// TIA Portal V20 export
ORGANIZATION_BLOCK "Startup"   // OB1020, LAD, Startup
TITLE = "Complete Restart"
AUTHOR : ERsystem_FA2_DH. Kim
// stored: AutoNumber false, IsIECCheckEnabled true, Namespace Unit1.Em2, SetENOAutomatically false
   VAR_INPUT
      LostRetentive : Bool;   // True if retentive data are lost
      LostRTC : Bool;   // True if date and time are lost
   END_VAR
BEGIN

REGION Network 1 (SCL): Build the Absolut Reference Designator
   // Set the Absoult Reference Designator in the Config DB
   IF LEN(IN := "Unit1.Em2.Config".em.referenceDesignator.parent) <> 0 THEN
     "Unit1.Em2.Config".em.referenceDesignator.combined := CONCAT_WSTRING(IN1 := "Unit1.Em2.Config".em.referenceDesignator.parent, IN2 := WSTRING#'.', IN3 := "Unit1.Em2.Config".em.referenceDesignator.relative);
   ELSE
     "Unit1.Em2.Config".em.referenceDesignator.combined := "Unit1.Em2.Config".em.referenceDesignator.relative;
   END_IF;
END_REGION

REGION Network 2 (SCL): Assign axes data
   //Assign axes
   // EM2 Have No Axis

   // Assign configuration data of axis
END_REGION

REGION Network 3 (SCL): Assign TwowayActuator Data
   //cmSuctionPadTopUpDown
   "Unit1.Em2.Config".cmSuctionPadTopUpDown.referenceDesignator := WSTRING#'cmSuctionPadTopUpDown';
   "Unit1.Em2.Config".cmSuctionPadTopUpDown.monitoringLeavingFeedback := T#1S;
   "Unit1.Em2.Config".cmSuctionPadTopUpDown.monitoringReachingFeedback := T#1S;
   "Unit1.Em2.Config".cmSuctionPadTopUpDown.disableFeedbackHomePos := FALSE;
   "Unit1.Em2.Config".cmSuctionPadTopUpDown.disableFeedbackWorkPos := FALSE;
   "Unit1.Em2.Config".cmSuctionPadTopUpDown.disableAlarms := FALSE;

   "Unit1.Em2.HmiInterface".cmSuctionPadTopUpDown.configuration.referenceDesignator := WSTRING#'cmSuctionPadTopUpDown';

   //cmSuctionPadBtmUpDown
   "Unit1.Em2.Config".cmSuctionPadBtmUpDown.referenceDesignator := WSTRING#'cmSuctionPadBtmUpDown';
   "Unit1.Em2.Config".cmSuctionPadBtmUpDown.monitoringLeavingFeedback := T#1S;
   "Unit1.Em2.Config".cmSuctionPadBtmUpDown.monitoringReachingFeedback := T#1S;
   "Unit1.Em2.Config".cmSuctionPadBtmUpDown.disableFeedbackHomePos := FALSE;
   "Unit1.Em2.Config".cmSuctionPadBtmUpDown.disableFeedbackWorkPos := FALSE;
   "Unit1.Em2.Config".cmSuctionPadBtmUpDown.disableAlarms := FALSE;

   "Unit1.Em2.HmiInterface".cmSuctionPadBtmUpDown.configuration.referenceDesignator := WSTRING#'cmSuctionPadBtmUpDown';

   //cmCutterUpDown
   "Unit1.Em2.Config".cmCutterUpDown.referenceDesignator := WSTRING#'cmCutterUpDown';
   "Unit1.Em2.Config".cmCutterUpDown.monitoringLeavingFeedback := T#1S;
   "Unit1.Em2.Config".cmCutterUpDown.monitoringReachingFeedback := T#1S;
   "Unit1.Em2.Config".cmCutterUpDown.disableFeedbackHomePos := FALSE;
   "Unit1.Em2.Config".cmCutterUpDown.disableFeedbackWorkPos := FALSE;
   "Unit1.Em2.Config".cmCutterUpDown.disableAlarms := FALSE;

   "Unit1.Em2.HmiInterface".cmCutterUpDown.configuration.referenceDesignator := WSTRING#'cmCutterUpDown';

   //cmTapeTopUpDown
   "Unit1.Em2.Config".cmTapeTopUpDown.referenceDesignator := WSTRING#'cmTapeTopUpDown';
   "Unit1.Em2.Config".cmTapeTopUpDown.monitoringLeavingFeedback := T#1S;
   "Unit1.Em2.Config".cmTapeTopUpDown.monitoringReachingFeedback := T#1S;
   "Unit1.Em2.Config".cmTapeTopUpDown.disableFeedbackHomePos := FALSE;
   "Unit1.Em2.Config".cmTapeTopUpDown.disableFeedbackWorkPos := FALSE;
   "Unit1.Em2.Config".cmTapeTopUpDown.disableAlarms := FALSE;

   "Unit1.Em2.HmiInterface".cmTapeTopUpDown.configuration.referenceDesignator := WSTRING#'cmTapeTopUpDown';

   //cmTapeBtmUpDown
   "Unit1.Em2.Config".cmTapeBtmUpDown.referenceDesignator := WSTRING#'cmTapeBtmUpDown';
   "Unit1.Em2.Config".cmTapeBtmUpDown.monitoringLeavingFeedback := T#1S;
   "Unit1.Em2.Config".cmTapeBtmUpDown.monitoringReachingFeedback := T#1S;
   "Unit1.Em2.Config".cmTapeBtmUpDown.disableFeedbackHomePos := FALSE;
   "Unit1.Em2.Config".cmTapeBtmUpDown.disableFeedbackWorkPos := FALSE;
   "Unit1.Em2.Config".cmTapeBtmUpDown.disableAlarms := FALSE;

   "Unit1.Em2.HmiInterface".cmTapeBtmUpDown.configuration.referenceDesignator := WSTRING#'cmTapeBtmUpDown';

   //cmSpliceHeadRotateTopFwdBwd
   "Unit1.Em2.Config".cmSpliceHeadRotateTopFwdBwd.referenceDesignator := WSTRING#'cmSpliceRotateTopFwdBwd';
   "Unit1.Em2.Config".cmSpliceHeadRotateTopFwdBwd.monitoringLeavingFeedback := T#1S;
   "Unit1.Em2.Config".cmSpliceHeadRotateTopFwdBwd.monitoringReachingFeedback := T#1S;
   "Unit1.Em2.Config".cmSpliceHeadRotateTopFwdBwd.disableFeedbackHomePos := FALSE;
   "Unit1.Em2.Config".cmSpliceHeadRotateTopFwdBwd.disableFeedbackWorkPos := FALSE;
   "Unit1.Em2.Config".cmSpliceHeadRotateTopFwdBwd.disableAlarms := FALSE;

   "Unit1.Em2.HmiInterface".cmSpliceHeadRotateTopFwdBwd.configuration.referenceDesignator := WSTRING#'cmSpliceRotateTopFwdBwd';

   //cmSpliceHeadRotateBtmFwdBwd
   "Unit1.Em2.Config".cmSpliceHeadRotateBtmFwdBwd.referenceDesignator := WSTRING#'cmSpliceRotateBtmFwdBwd';
   "Unit1.Em2.Config".cmSpliceHeadRotateBtmFwdBwd.monitoringLeavingFeedback := T#1S;
   "Unit1.Em2.Config".cmSpliceHeadRotateBtmFwdBwd.monitoringReachingFeedback := T#1S;
   "Unit1.Em2.Config".cmSpliceHeadRotateBtmFwdBwd.disableFeedbackHomePos := FALSE;
   "Unit1.Em2.Config".cmSpliceHeadRotateBtmFwdBwd.disableFeedbackWorkPos := FALSE;
   "Unit1.Em2.Config".cmSpliceHeadRotateBtmFwdBwd.disableAlarms := FALSE;

   "Unit1.Em2.HmiInterface".cmSpliceHeadRotateBtmFwdBwd.configuration.referenceDesignator := WSTRING#'cmSpliceRotateBtmFwdBwd';

   //cmSuctionPadTopLeftVaccum
   "Unit1.Em2.Config".cmSuctionPadTopLeftVaccum.referenceDesignator := WSTRING#'cmSuctionPadTopLeftVac';
   "Unit1.Em2.Config".cmSuctionPadTopLeftVaccum.monitoringLeavingFeedback := T#1S;
   "Unit1.Em2.Config".cmSuctionPadTopLeftVaccum.monitoringReachingFeedback := T#1S;
   "Unit1.Em2.Config".cmSuctionPadTopLeftVaccum.disableFeedbackHomePos := FALSE;
   "Unit1.Em2.Config".cmSuctionPadTopLeftVaccum.disableFeedbackWorkPos := FALSE;
   "Unit1.Em2.Config".cmSuctionPadTopLeftVaccum.disableAlarms := FALSE;

   "Unit1.Em2.HmiInterface".cmSuctionPadTopLeftVaccum.configuration.referenceDesignator := WSTRING#'cmSuctionPadTopLeftVac';

   //cmSuctionPadTopRightVaccum
   "Unit1.Em2.Config".cmSuctionPadTopRightVaccum.referenceDesignator := WSTRING#'cmSuctionPadTopRightVac';
   "Unit1.Em2.Config".cmSuctionPadTopRightVaccum.monitoringLeavingFeedback := T#1S;
   "Unit1.Em2.Config".cmSuctionPadTopRightVaccum.monitoringReachingFeedback := T#1S;
   "Unit1.Em2.Config".cmSuctionPadTopRightVaccum.disableFeedbackHomePos := FALSE;
   "Unit1.Em2.Config".cmSuctionPadTopRightVaccum.disableFeedbackWorkPos := FALSE;
   "Unit1.Em2.Config".cmSuctionPadTopRightVaccum.disableAlarms := FALSE;

   "Unit1.Em2.HmiInterface".cmSuctionPadTopRightVaccum.configuration.referenceDesignator := WSTRING#'cmSuctionPadTopRightVac';

   //cmSuctionPadBtmLeftVaccum
   "Unit1.Em2.Config".cmSuctionPadBtmLeftVaccum.referenceDesignator := WSTRING#'cmSuctionPadBtmLeftVac';
   "Unit1.Em2.Config".cmSuctionPadBtmLeftVaccum.monitoringLeavingFeedback := T#1S;
   "Unit1.Em2.Config".cmSuctionPadBtmLeftVaccum.monitoringReachingFeedback := T#1S;
   "Unit1.Em2.Config".cmSuctionPadBtmLeftVaccum.disableFeedbackHomePos := FALSE;
   "Unit1.Em2.Config".cmSuctionPadBtmLeftVaccum.disableFeedbackWorkPos := FALSE;
   "Unit1.Em2.Config".cmSuctionPadBtmLeftVaccum.disableAlarms := FALSE;

   "Unit1.Em2.HmiInterface".cmSuctionPadBtmLeftVaccum.configuration.referenceDesignator := WSTRING#'cmSuctionPadBtmLeftVac';

   //cmSuctionPadBtmRightVaccum
   "Unit1.Em2.Config".cmSuctionPadBtmRightVaccum.referenceDesignator := WSTRING#'cmSuctionPadBtmRightVac';
   "Unit1.Em2.Config".cmSuctionPadBtmRightVaccum.monitoringLeavingFeedback := T#1S;
   "Unit1.Em2.Config".cmSuctionPadBtmRightVaccum.monitoringReachingFeedback := T#1S;
   "Unit1.Em2.Config".cmSuctionPadBtmRightVaccum.disableFeedbackHomePos := FALSE;
   "Unit1.Em2.Config".cmSuctionPadBtmRightVaccum.disableFeedbackWorkPos := FALSE;
   "Unit1.Em2.Config".cmSuctionPadBtmRightVaccum.disableAlarms := FALSE;

   "Unit1.Em2.HmiInterface".cmSuctionPadBtmRightVaccum.configuration.referenceDesignator := WSTRING#'cmSuctionPadBtmRightVac';

   //cmSuctionPadTopTapeVaccum
   "Unit1.Em2.Config".cmSuctionPadTopTapeVaccum.referenceDesignator := WSTRING#'cmSuctionPadTopTapeVac';
   "Unit1.Em2.Config".cmSuctionPadTopTapeVaccum.monitoringLeavingFeedback := T#1S;
   "Unit1.Em2.Config".cmSuctionPadTopTapeVaccum.monitoringReachingFeedback := T#1S;
   "Unit1.Em2.Config".cmSuctionPadTopTapeVaccum.disableFeedbackHomePos := FALSE;
   "Unit1.Em2.Config".cmSuctionPadTopTapeVaccum.disableFeedbackWorkPos := FALSE;
   "Unit1.Em2.Config".cmSuctionPadTopTapeVaccum.disableAlarms := FALSE;

   "Unit1.Em2.HmiInterface".cmSuctionPadTopTapeVaccum.configuration.referenceDesignator := WSTRING#'cmSuctionPadTopTapeVac';

   //cmSuctionPadBtmTapeVaccum
   "Unit1.Em2.Config".cmSuctionPadBtmTapeVaccum.referenceDesignator := WSTRING#'cmSuctionPadBtmTapeVac';
   "Unit1.Em2.Config".cmSuctionPadBtmTapeVaccum.monitoringLeavingFeedback := T#1S;
   "Unit1.Em2.Config".cmSuctionPadBtmTapeVaccum.monitoringReachingFeedback := T#1S;
   "Unit1.Em2.Config".cmSuctionPadBtmTapeVaccum.disableFeedbackHomePos := FALSE;
   "Unit1.Em2.Config".cmSuctionPadBtmTapeVaccum.disableFeedbackWorkPos := FALSE;
   "Unit1.Em2.Config".cmSuctionPadBtmTapeVaccum.disableAlarms := FALSE;

   "Unit1.Em2.HmiInterface".cmSuctionPadBtmTapeVaccum.configuration.referenceDesignator := WSTRING#'cmSuctionPadBtmTapeVac';
END_REGION
END_ORGANIZATION_BLOCK
